Staubli VAL3: stop.pgx

program stop()
begin
  //
  // QUIT KERNEL
  //
  call kernel:stop()
  cls()
end
